{attribute 'GeneratedUsingTerminal: EL1512-0000-0017'}
{attribute addProperty BoxType "EL1512-0000-0017"}
{attribute addProperty Id "Set_counterBOOL1Inhibit_counterBOOL1"}
{attribute addProperty CRC "187665264"}
{attribute addProperty Size "2"}
TYPE Control_0B2F8B70 :
STRUCT
	{attribute addProperty Name "Set_counter"}
	Set_counter : BOOL;
	{attribute addProperty Name "Inhibit_counter"}
	Inhibit_counter : BOOL;
END_STRUCT
END_TYPE

(* stored: Version 1.2.0.0, ProductVersion 3.1.4024.9
   DUT Control_0B2F8B70: Id {d5e726a8-176c-4b53-8321-a620642dc030} *)
